TYPE SmotorParameter :
STRUCT
	max_speed : REAL := 100;
	min_speed : REAL := 1;
END_STRUCT
END_TYPE

(* stored: Version 1.1.0.1, ProductVersion 3.1.4024.12
   DUT SmotorParameter: Id {a754dd86-52cb-4da6-805a-8eff512fd6cd} *)
